TYPE st_ConnectionInfoData :
STRUCT
	state,diag:USINT;
	bit1,bit2,bit3,bit4:BIT;
END_STRUCT
END_TYPE

(* stored: Version 1.1.0.1, ProductVersion 3.1.4024.12
   DUT st_ConnectionInfoData: Id {23ae5872-e503-47b7-9ef2-35e94bca9d76} *)
